FUNCTION_BLOCK CmdOneAct (* CAT Function Block Type *)
  (* Standard: 61499-2 *)
  (* Version 0.0, 6/7/2026, Schneider Electric, template *)
  PACKAGE SE.Nereda;
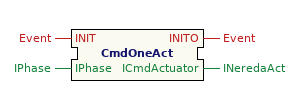
  EVENT_INPUT
    INIT;
  END_EVENT
  EVENT_OUTPUT
    INITO;
  END_EVENT
  SOCKETS
    IPhase : IPhase;
  END_SOCKETS
  PLUGS
    ICmdActuator : INeredaAct;
  END_PLUGS
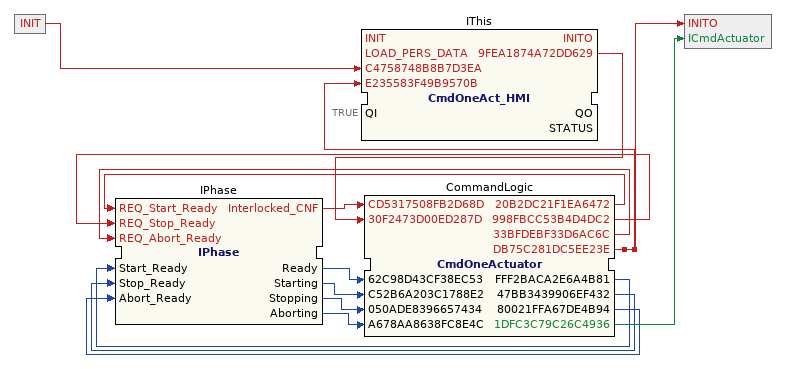
  (* 01 - FUNCTIONNAL INPUT INTERFACE *)
  (* 00 - INITIALIZATION *)
  (* 05 - LOGIC *)
  (* 06 - HMI INTERFACE *)
  (* 03 - FIELD INTERFACE *)
  (* 02 - FUNCTIONNAL OUTPUT INTERFACE *)
  (* Command Logic *)
  FBS
    IThis : CmdOneAct_HMI(QI := TRUE);
    CommandLogic : CmdOneActuator; {SET_ATTRIBUTE(Configuration.Component.HideUnusedPorts, )}
  END_FBS
  EVENT_CONNECTIONS
    INIT TO IThis.C4758748B8B7D3EA;
    IPhase.Interlocked_CNF TO CommandLogic.CD5317508FB2D68D;
    IThis.9FEA1874A72DD629 TO CommandLogic.30F2473D00ED287D;
    CommandLogic.20B2DC21F1EA6472 TO IPhase.REQ_Start_Ready;
    CommandLogic.998FBCC53B4D4DC2 TO IPhase.REQ_Stop_Ready;
    CommandLogic.33BFDEBF33D6AC6C TO IPhase.REQ_Abort_Ready;
    CommandLogic.DB75C281DC5EE23E TO INITO;
    CommandLogic.DB75C281DC5EE23E TO IThis.E235583F49B9570B;
  END_CONNECTIONS
  DATA_CONNECTIONS
    IPhase.Ready TO CommandLogic.62C98D43CF38EC53;
    IPhase.Starting TO CommandLogic.C52B6A203C1788E2;
    IPhase.Stopping TO CommandLogic.050ADE8396657434;
    IPhase.Aborting TO CommandLogic.A678AA8638FC8E4C;
    CommandLogic.FFF2BACA2E6A4B81 TO IPhase.Start_Ready;
    CommandLogic.47BB3439906EF432 TO IPhase.Stop_Ready;
    CommandLogic.80021FFA67DE4B94 TO IPhase.Abort_Ready;
  END_CONNECTIONS
  ADAPTER_CONNECTIONS
    CommandLogic.1DFC3C79C26C4936 TO ICmdActuator;
  END_CONNECTIONS
END_FUNCTION_BLOCK
